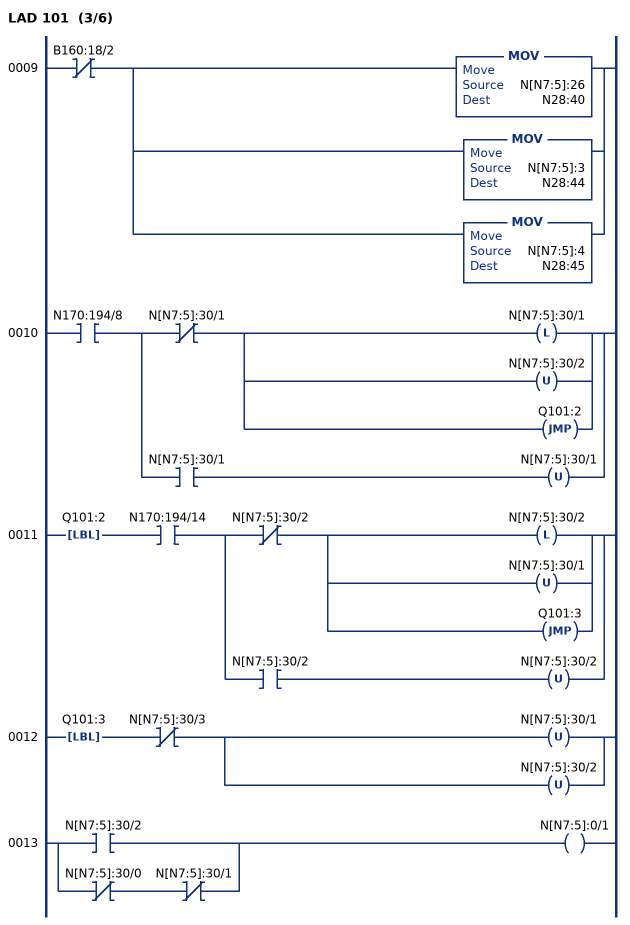
% Rung: 9 %
SOR XIO B160:18/2 BST MOV N[N7:5]:26 N28:40 NXB MOV N[N7:5]:3 N28:44 NXB MOV N[N7:5]:4 N28:45 BND EOR
% Rung: 10 %
SOR XIC N170:194/8 BST XIO N[N7:5]:30/1 BST OTL N[N7:5]:30/1 NXB OTU N[N7:5]:30/2 NXB JMP Q101:2 BND NXB XIC N[N7:5]:30/1 OTU N[N7:5]:30/1 BND EOR
% Rung: 11 %
SOR LBL Q101:2 XIC N170:194/14 BST XIO N[N7:5]:30/2 BST OTL N[N7:5]:30/2 NXB OTU N[N7:5]:30/1 NXB JMP Q101:3 BND NXB XIC N[N7:5]:30/2 OTU N[N7:5]:30/2 BND EOR
% Rung: 12 %
SOR LBL Q101:3 XIO N[N7:5]:30/3 BST OTU N[N7:5]:30/1 NXB OTU N[N7:5]:30/2 BND EOR
% Rung: 13 %
SOR BST XIC N[N7:5]:30/2 NXB XIO N[N7:5]:30/0 XIO N[N7:5]:30/1 BND OTE N[N7:5]:0/1 EOR

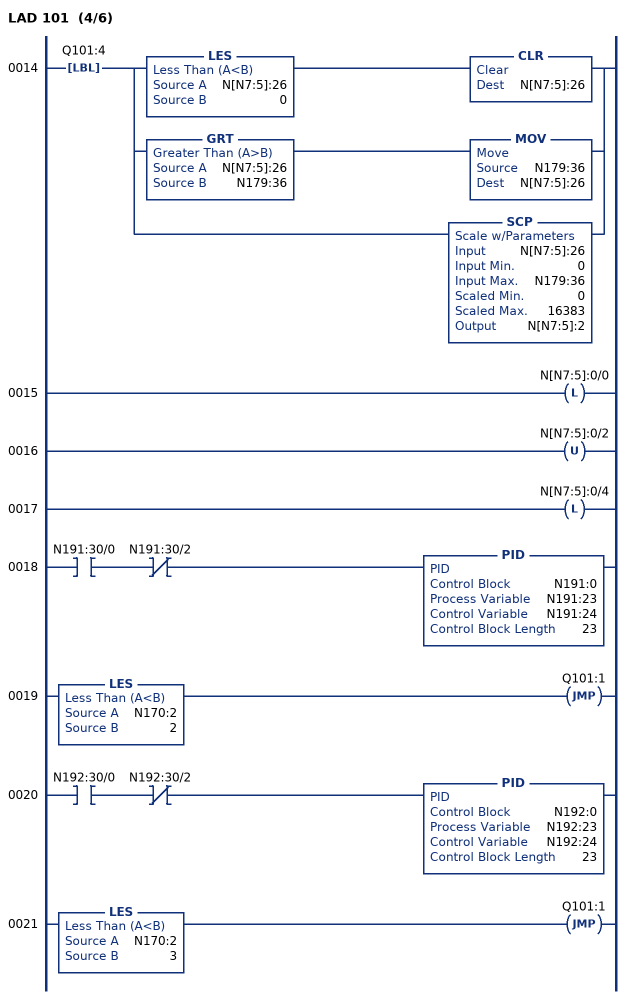
% Rung: 14 %
SOR LBL Q101:4 BST LES N[N7:5]:26 0 CLR N[N7:5]:26 NXB GRT N[N7:5]:26 N179:36 MOV N179:36 N[N7:5]:26 NXB SCP N[N7:5]:26 0 N179:36 0 16383 N[N7:5]:2 BND EOR
% Rung: 15 %
SOR OTL N[N7:5]:0/0 EOR
% Rung: 16 %
SOR OTU N[N7:5]:0/2 EOR
% Rung: 17 %
SOR OTL N[N7:5]:0/4 EOR
% Rung: 18 %
SOR XIC N191:30/0 XIO N191:30/2 PID N191:0 N191:23 N191:24 23 EOR
% Rung: 19 %
SOR LES N170:2 2 JMP Q101:1 EOR
% Rung: 20 %
SOR XIC N192:30/0 XIO N192:30/2 PID N192:0 N192:23 N192:24 23 EOR
% Rung: 21 %
SOR LES N170:2 3 JMP Q101:1 EOR

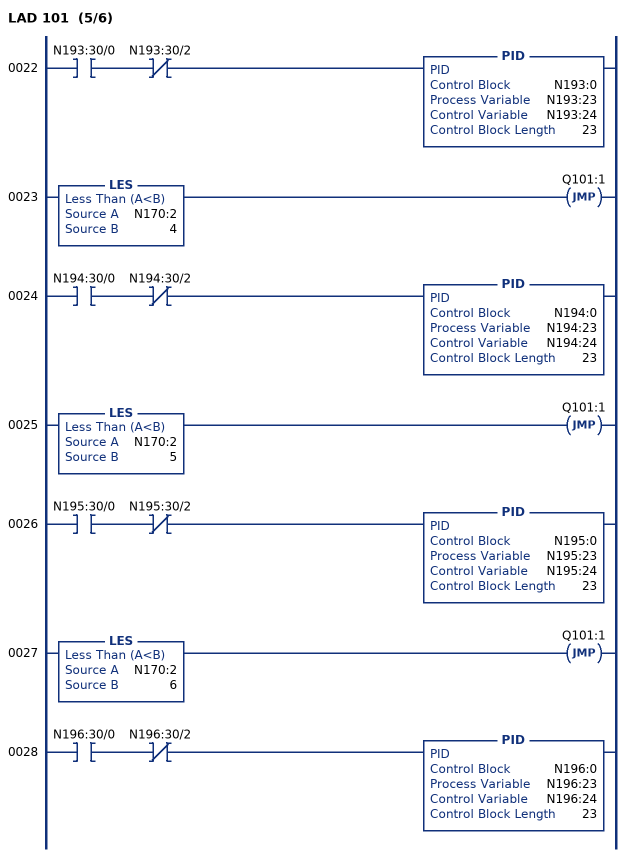
% Rung: 22 %
SOR XIC N193:30/0 XIO N193:30/2 PID N193:0 N193:23 N193:24 23 EOR
% Rung: 23 %
SOR LES N170:2 4 JMP Q101:1 EOR
% Rung: 24 %
SOR XIC N194:30/0 XIO N194:30/2 PID N194:0 N194:23 N194:24 23 EOR
% Rung: 25 %
SOR LES N170:2 5 JMP Q101:1 EOR
% Rung: 26 %
SOR XIC N195:30/0 XIO N195:30/2 PID N195:0 N195:23 N195:24 23 EOR
% Rung: 27 %
SOR LES N170:2 6 JMP Q101:1 EOR
% Rung: 28 %
SOR XIC N196:30/0 XIO N196:30/2 PID N196:0 N196:23 N196:24 23 EOR

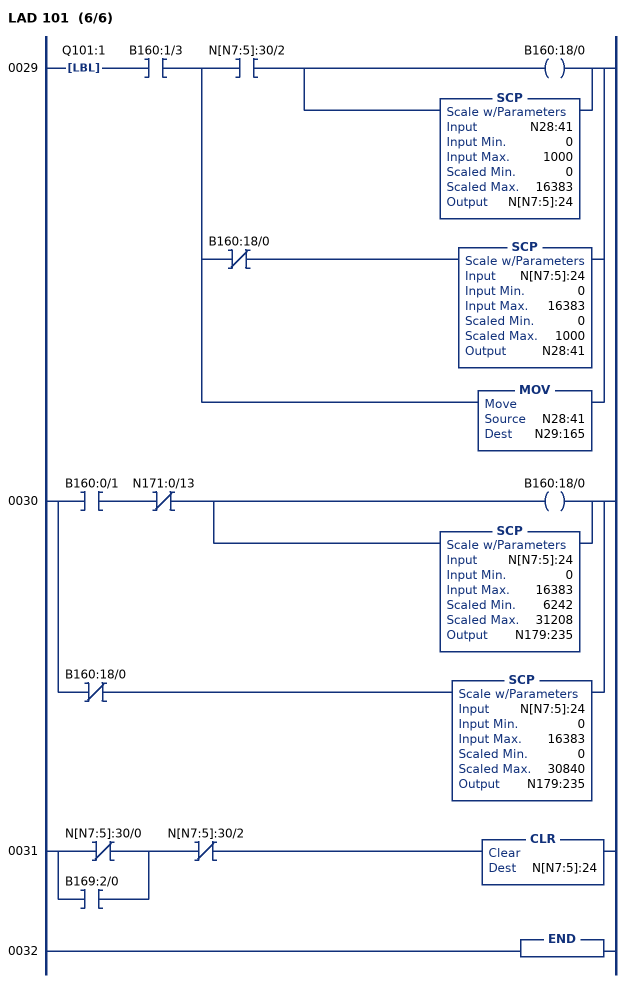
% Rung: 29 %
SOR LBL Q101:1 XIC B160:1/3 BST XIC N[N7:5]:30/2 BST OTE B160:18/0 NXB SCP N28:41 0 1000 0 16383 N[N7:5]:24 BND NXB XIO B160:18/0 SCP N[N7:5]:24 0 16383 0 1000 N28:41 NXB MOV N28:41 N29:165 BND EOR
% Rung: 30 %
SOR BST XIC B160:0/1 XIO N171:0/13 BST OTE B160:18/0 NXB SCP N[N7:5]:24 0 16383 6242 31208 N179:235 BND NXB XIO B160:18/0 SCP N[N7:5]:24 0 16383 0 30840 N179:235 BND EOR
% Rung: 31 %
SOR BST XIO N[N7:5]:30/0 NXB XIC B169:2/0 BND XIO N[N7:5]:30/2 CLR N[N7:5]:24 EOR
% Rung: 32 %
SOR END EOR

LADDER 102
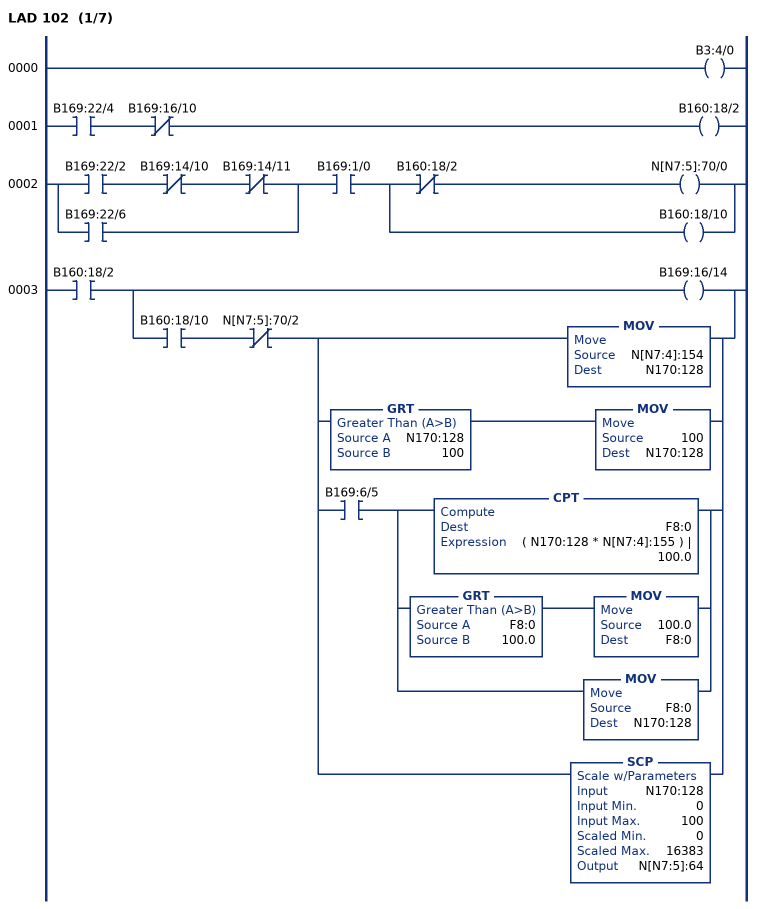
% Rung: 0 %
SOR OTE B3:4/0 EOR
% Rung: 1 %
SOR XIC B169:22/4 XIO B169:16/10 OTE B160:18/2 EOR
% Rung: 2 %
SOR BST XIC B169:22/2 XIO B169:14/10 XIO B169:14/11 NXB XIC B169:22/6 BND XIC B169:1/0 BST XIO B160:18/2 OTE N[N7:5]:70/0 NXB OTE B160:18/10 BND EOR
% Rung: 3 %
SOR XIC B160:18/2 BST OTE B169:16/14 NXB XIC B160:18/10 XIO N[N7:5]:70/2 BST BST MOV N[N7:4]:154 N170:128 NXB GRT N170:128 100 MOV 100 N170:128 BND NXB XIC B169:6/5 BST CPT F8:0 " ( N170:128 * N[N7:4]:155 ) | 100.0 " NXB GRT F8:0 100.0 MOV 100.0 F8:0 NXB MOV F8:0 N170:128 BND NXB SCP N170:128 0 100 0 16383 N[N7:5]:64 BND BND EOR

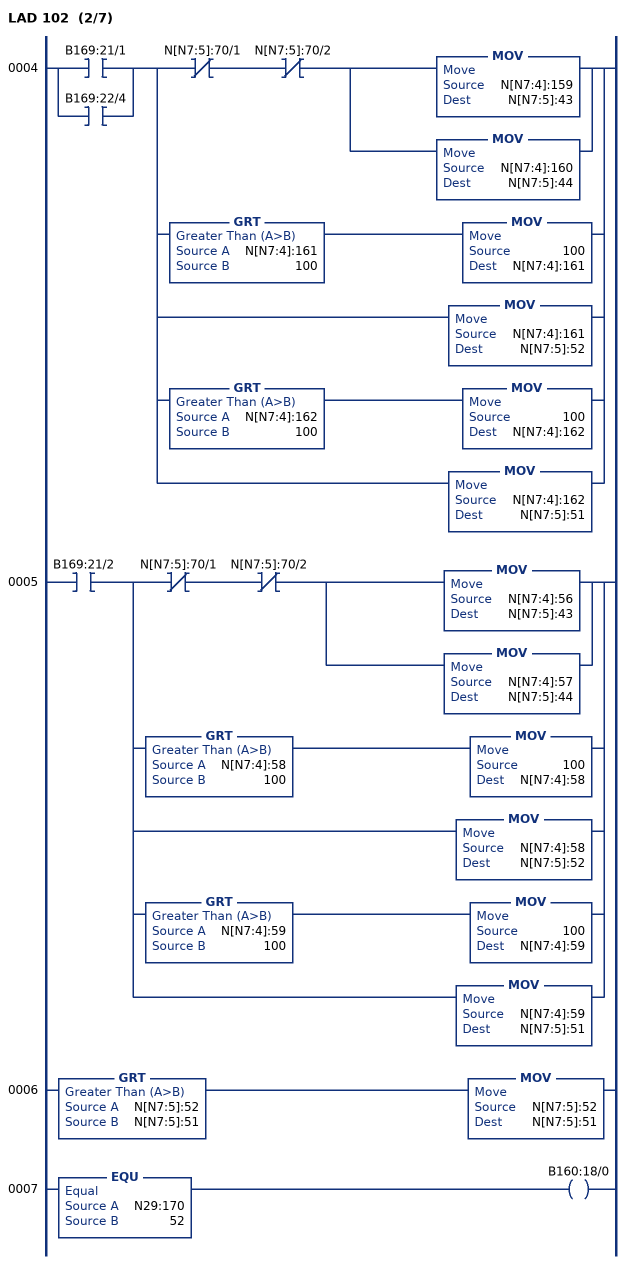
% Rung: 4 %
SOR BST XIC B169:21/1 NXB XIC B169:22/4 BND BST XIO N[N7:5]:70/1 XIO N[N7:5]:70/2 BST MOV N[N7:4]:159 N[N7:5]:43 NXB MOV N[N7:4]:160 N[N7:5]:44 BND NXB GRT N[N7:4]:161 100 MOV 100 N[N7:4]:161 NXB MOV N[N7:4]:161 N[N7:5]:52 NXB GRT N[N7:4]:162 100 MOV 100 N[N7:4]:162 NXB MOV N[N7:4]:162 N[N7:5]:51 BND EOR
% Rung: 5 %
SOR XIC B169:21/2 BST XIO N[N7:5]:70/1 XIO N[N7:5]:70/2 BST MOV N[N7:4]:56 N[N7:5]:43 NXB MOV N[N7:4]:57 N[N7:5]:44 BND NXB GRT N[N7:4]:58 100 MOV 100 N[N7:4]:58 NXB MOV N[N7:4]:58 N[N7:5]:52 NXB GRT N[N7:4]:59 100 MOV 100 N[N7:4]:59 NXB MOV N[N7:4]:59 N[N7:5]:51 BND EOR
% Rung: 6 %
SOR GRT N[N7:5]:52 N[N7:5]:51 MOV N[N7:5]:52 N[N7:5]:51 EOR
% Rung: 7 %
SOR EQU N29:170 52 OTE B160:18/0 EOR

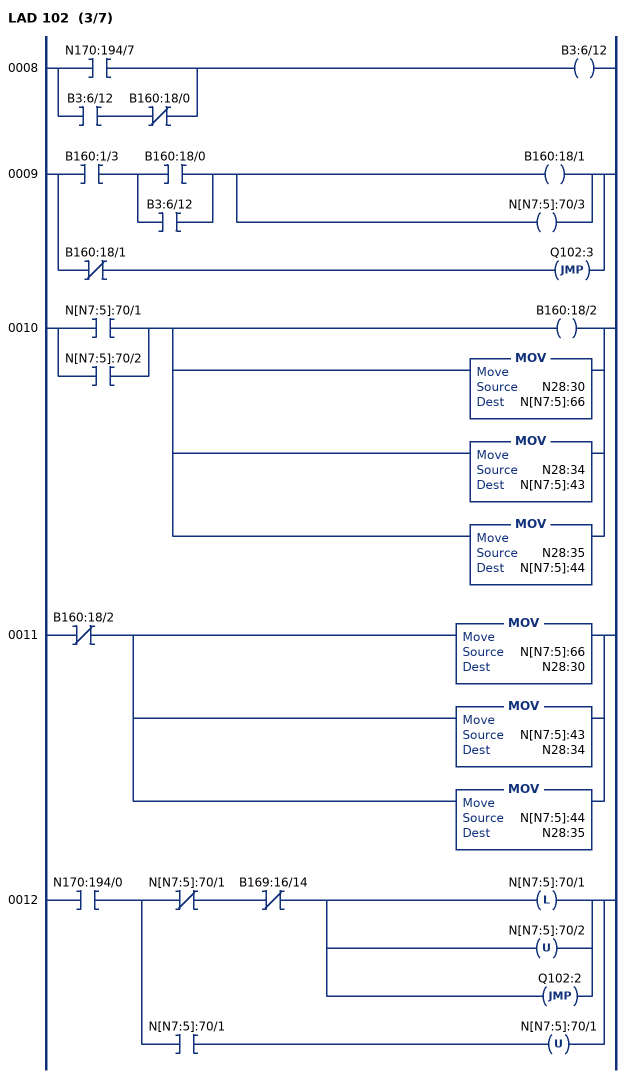
% Rung: 8 %
SOR BST XIC N170:194/7 NXB XIC B3:6/12 XIO B160:18/0 BND OTE B3:6/12 EOR
% Rung: 9 %
SOR BST XIC B160:1/3 BST XIC B160:18/0 NXB XIC B3:6/12 BND BST OTE B160:18/1 NXB OTE N[N7:5]:70/3 BND NXB XIO B160:18/1 JMP Q102:3 BND EOR
% Rung: 10 %
SOR BST XIC N[N7:5]:70/1 NXB XIC N[N7:5]:70/2 BND BST OTE B160:18/2 NXB MOV N28:30 N[N7:5]:66 NXB MOV N28:34 N[N7:5]:43 NXB MOV N28:35 N[N7:5]:44 BND EOR
% Rung: 11 %
SOR XIO B160:18/2 BST MOV N[N7:5]:66 N28:30 NXB MOV N[N7:5]:43 N28:34 NXB MOV N[N7:5]:44 N28:35 BND EOR
% Rung: 12 %
SOR XIC N170:194/0 BST XIO N[N7:5]:70/1 XIO B169:16/14 BST OTL N[N7:5]:70/1 NXB OTU N[N7:5]:70/2 NXB JMP Q102:2 BND NXB XIC N[N7:5]:70/1 OTU N[N7:5]:70/1 BND EOR

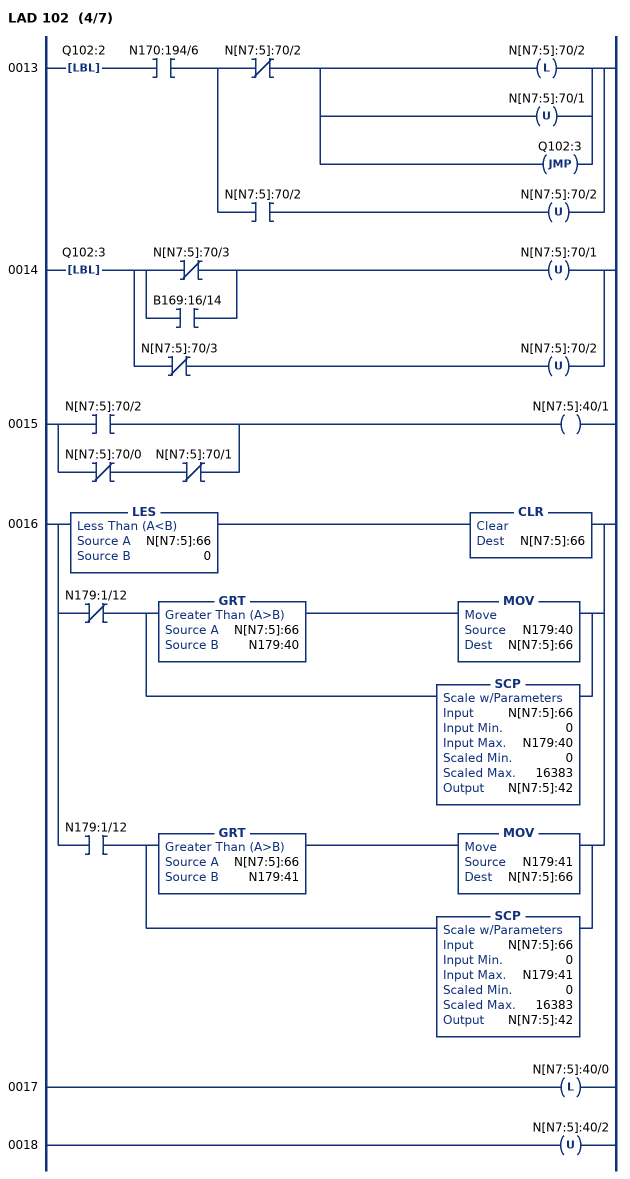
% Rung: 13 %
SOR LBL Q102:2 XIC N170:194/6 BST XIO N[N7:5]:70/2 BST OTL N[N7:5]:70/2 NXB OTU N[N7:5]:70/1 NXB JMP Q102:3 BND NXB XIC N[N7:5]:70/2 OTU N[N7:5]:70/2 BND EOR
% Rung: 14 %
SOR LBL Q102:3 BST BST XIO N[N7:5]:70/3 NXB XIC B169:16/14 BND OTU N[N7:5]:70/1 NXB XIO N[N7:5]:70/3 OTU N[N7:5]:70/2 BND EOR
% Rung: 15 %
SOR BST XIC N[N7:5]:70/2 NXB XIO N[N7:5]:70/0 XIO N[N7:5]:70/1 BND OTE N[N7:5]:40/1 EOR
% Rung: 16 %
SOR BST LES N[N7:5]:66 0 CLR N[N7:5]:66 NXB XIO N179:1/12 BST GRT N[N7:5]:66 N179:40 MOV N179:40 N[N7:5]:66 NXB SCP N[N7:5]:66 0 N179:40 0 16383 N[N7:5]:42 BND NXB XIC N179:1/12 BST GRT N[N7:5]:66 N179:41 MOV N179:41 N[N7:5]:66 NXB SCP N[N7:5]:66 0 N179:41 0 16383 N[N7:5]:42 BND BND EOR
% Rung: 17 %
SOR OTL N[N7:5]:40/0 EOR
% Rung: 18 %
SOR OTU N[N7:5]:40/2 EOR

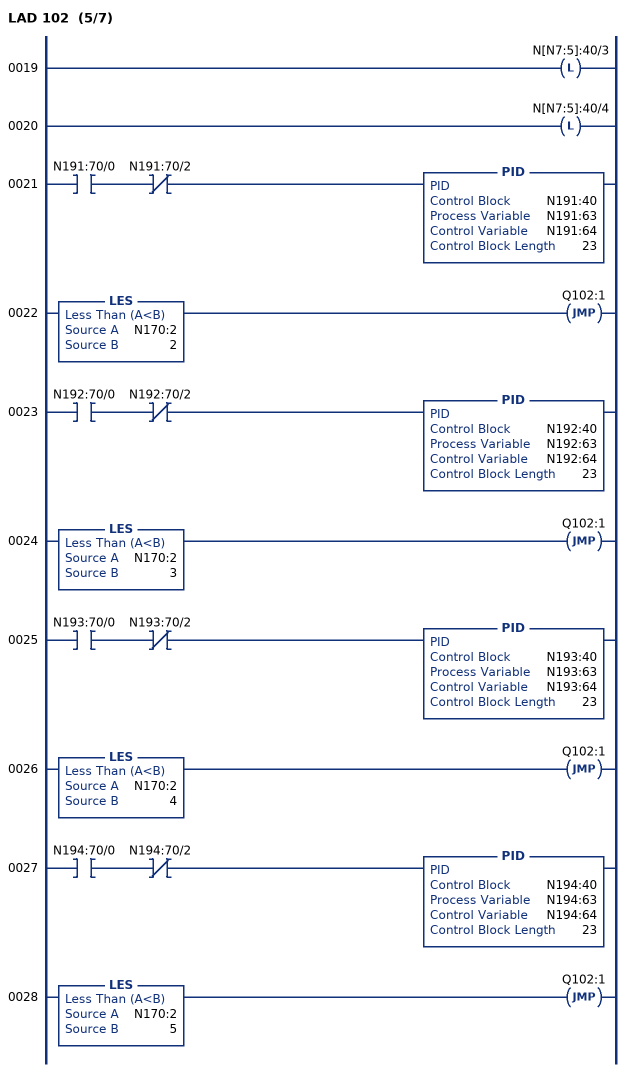
% Rung: 19 %
SOR OTL N[N7:5]:40/3 EOR
% Rung: 20 %
SOR OTL N[N7:5]:40/4 EOR
% Rung: 21 %
SOR XIC N191:70/0 XIO N191:70/2 PID N191:40 N191:63 N191:64 23 EOR
% Rung: 22 %
SOR LES N170:2 2 JMP Q102:1 EOR
% Rung: 23 %
SOR XIC N192:70/0 XIO N192:70/2 PID N192:40 N192:63 N192:64 23 EOR
% Rung: 24 %
SOR LES N170:2 3 JMP Q102:1 EOR
% Rung: 25 %
SOR XIC N193:70/0 XIO N193:70/2 PID N193:40 N193:63 N193:64 23 EOR
% Rung: 26 %
SOR LES N170:2 4 JMP Q102:1 EOR
% Rung: 27 %
SOR XIC N194:70/0 XIO N194:70/2 PID N194:40 N194:63 N194:64 23 EOR
% Rung: 28 %
SOR LES N170:2 5 JMP Q102:1 EOR

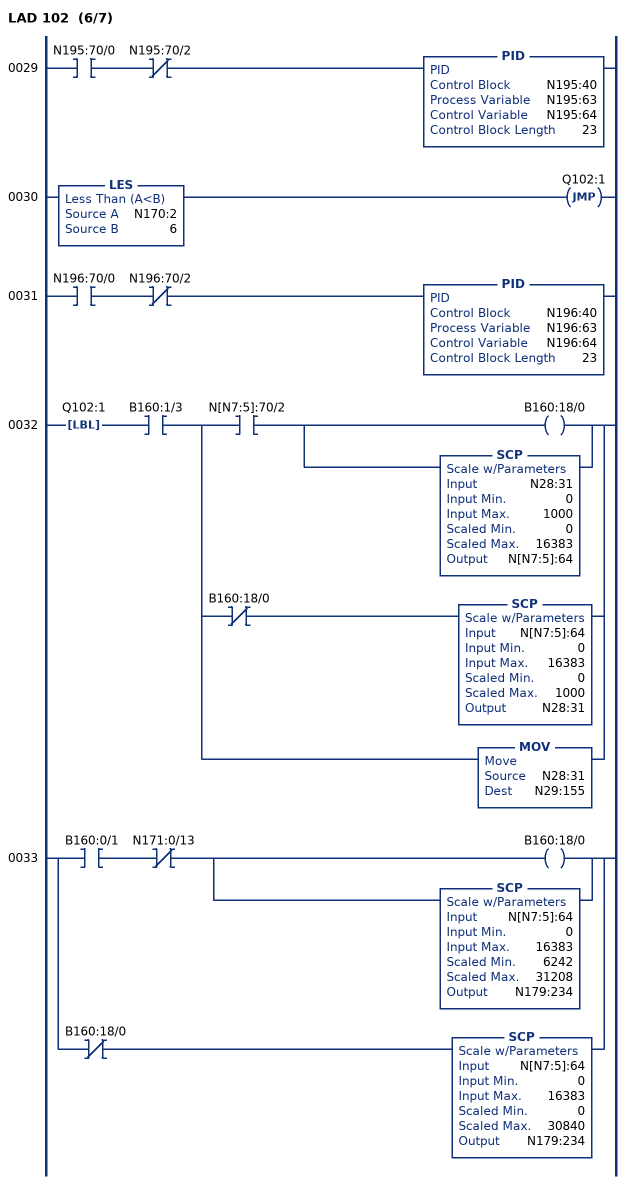
% Rung: 29 %
SOR XIC N195:70/0 XIO N195:70/2 PID N195:40 N195:63 N195:64 23 EOR
% Rung: 30 %
SOR LES N170:2 6 JMP Q102:1 EOR
% Rung: 31 %
SOR XIC N196:70/0 XIO N196:70/2 PID N196:40 N196:63 N196:64 23 EOR
% Rung: 32 %
SOR LBL Q102:1 XIC B160:1/3 BST XIC N[N7:5]:70/2 BST OTE B160:18/0 NXB SCP N28:31 0 1000 0 16383 N[N7:5]:64 BND NXB XIO B160:18/0 SCP N[N7:5]:64 0 16383 0 1000 N28:31 NXB MOV N28:31 N29:155 BND EOR
% Rung: 33 %
SOR BST XIC B160:0/1 XIO N171:0/13 BST OTE B160:18/0 NXB SCP N[N7:5]:64 0 16383 6242 31208 N179:234 BND NXB XIO B160:18/0 SCP N[N7:5]:64 0 16383 0 30840 N179:234 BND EOR

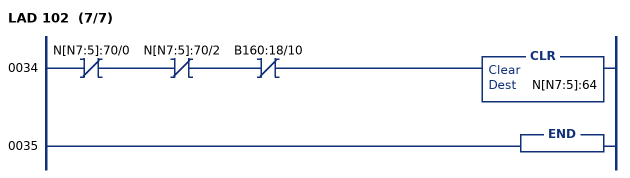
% Rung: 34 %
SOR XIO N[N7:5]:70/0 XIO N[N7:5]:70/2 XIO B160:18/10 CLR N[N7:5]:64 EOR
% Rung: 35 %
SOR END EOR

DATA TABLE (non-zero values as saved)
DATA B3
% B3:0 % 0X0802 0X0000 0X0200 0X0000 0X0009 0X0084 0X8000 0X0000 0X0040 0X0000
% B3:10 % 0X0000 0X0000 0X0000 0X0000 0X0000 0X0000 0X0000 0X0001
DATA T4
% .PRE .ACC %
% T4:2 % 5 5
% T4:3 % 5 0
% T4:9 % 60 0
% T4:10 % 2 0
% T4:11 % 3 0
% T4:15 % 5 0
% T4:19 % 1 0
% T4:20 % 1200 0
% T4:21 % 15 0
% T4:22 % 15 0
% T4:23 % 15 0
% T4:24 % 3 0
% T4:25 % 3 0
% T4:26 % 3 0
% T4:27 % 2 0
% T4:28 % 2 0
% T4:30 % 50 50
% T4:31 % 50 50
% T4:32 % 50 50
% T4:33 % 15 0
% T4:34 % 15 0
% T4:35 % 110 0
% T4:36 % 20 0
DATA C5
% .PRE .ACC %
% C5:5 % 3 0
DATA R6
% .LEN .POS %
% R6:0 % 16 0
% R6:1 % 10 0
% R6:2 % 10 0
% R6:3 % 10 0
% R6:4 % 10 0
% R6:5 % 10 0
% R6:6 % 10 0
% R6:7 % 11 0
% R6:8 % 8 0
% R6:9 % 16 0
% R6:11 % 10 10
% R6:12 % 10 10
% R6:13 % 10 0
% R6:14 % 10 0
% R6:15 % 10 0
% R6:16 % 10 0
% R6:17 % 32 0
% R6:18 % 6 0
% R6:19 % 6 0
% R6:20 % 32 0
DATA N7
% N7:0 % 2 162 172 182 60 192 202 212 232 0
% N7:10 % 41 1 166 0 0 0 0 0 0 0
% N7:20 % 3 5 1 0 0 0 0 0 0 0
% N7:30 % 0 8 0 2 0 -32768 0 0 0 0
% N7:40 % -32768 0 0 0 0 0 0 0 0 0
% N7:60 % 0 2 0 0 0 0 0 0 0 0
% N7:100 % 150 41 40 63 100 0 41 10 0 0
% N7:110 % 44 0 63 0 0 0 38 1 38 1
% N7:120 % 0 38 1 0 3 15 3 40 70 100
% N7:130 % 0 0 0 -1 0
DATA T10
% .PRE .ACC %
% T10:0 % 12 0
% T10:1 % 12 0
% T10:2 % 12 0
% T10:3 % 3 0
DATA N11
% N11:0 % 0 1 4 21 31 0 0 0 0 0
% N11:10 % 0 81 91 0 0 0 1 4 0 0
% N11:20 % 41 51 0 0 0 0 81 91 0 0
% N11:30 % 0 1 4 21 31 41 51 0 0 0
% N11:40 % 0 81 91 0 0 0 1 4 0 0
% N11:50 % 41 51 21 31 0 0 81 91 0 0
% N11:60 % 0 1 4 21 31 41 51 21 31 0
% N11:70 % 0 81 91 0 0 0 1 4 21 31
% N11:80 % 0 0 0 0 61 0 81 91 0 0
% N11:90 % 0 1 4 21 31 41 51 0 0 61
% N11:100 % 0 81 91 0 0 0 1 4 0 0
% N11:110 % 41 51 21 31 61 0 81 91 0 0
% N11:120 % 0 1 4 21 31 0 0 0 0 0
% N11:130 % 71 153 91 0 0 0 1 4 21 31
% N11:140 % 41 51 0 0 0 71 153 91 0 0
% N11:160 % 71 91 0 0 0 0 1 4 0 0
% N11:170 % 0 0 0 0 0 0 81 91 0 0
% N11:190 % 71 153 91 0 0 0 0 0 0 0
% N11:200 % 0 0 0 0 61 0 81 91 0 0
DATA N12
% N12:0 % 0 101 105 135 0 0 101 125 135 0
% N12:10 % 0 101 141 135 0 0 101 115 135 0
% N12:20 % 0 101 127 135 0 0 101 161 135 0
% N12:30 % 0 101 129 135 0 0 101 181 135 0
% N12:40 % 0 101 201 135 0 0 101 131 135 0
% N12:50 % 0 101 195 135 0
DATA N14
% N14:0 % 0 8193 0 0 8192 8240 8192 8240 48 0
% N14:10 % 528 562 34 1 48 34 0 0 0 0
% N14:20 % 0 1 40 0 40 2088 2600 -30174 2602 2082
% N14:30 % 0 2049 0 -30688 2048 -30688 -30688 -28640 -32222 4130
% N14:40 % 0 1 36 0 36 1060 1572 -31198 1574 1058
% N14:50 % 0 1025 0 -31712 1024 -31712 -31712 -28640 -32222 4130
% N14:60 % 0 1 -32736 0 -32736 -32224 -32222 2 0 0
% N14:70 % 0 2 32 0 32 544 0 546 34 0
% N14:80 % 0 1 0 -28640 4096 -28640 -28640 -28640 0 0
% N14:90 % 0 4096 0 0 0 0 0 0 0 0
% N14:100 % 0 193 0 0 0 -30496 2281 2280 2280 2280
% N14:110 % 2280 -30528 0 0 0 -31520 1253 1252 1252 1252
% N14:120 % 1252 -31552 0 0 0 200 0 196 0 208
% N14:130 % 0 192 0 0 0 -32640 -32576 0 0 0
% N14:140 % 0 2256 456 200 132 2276 488 201 -32640 -30528
% N14:150 % 456 201 0 1 -32768 0 -32768 -32768 -32254 2
% N14:160 % 0 1232 452 196 136 1256 484 197 -32640 -31552
% N14:170 % 452 197 0 0 0 0 0 0 0 0
% N14:180 % 0 -28480 464 208 136 4328 496 209 -32640 -28480
% N14:190 % 464 209 0 0 0 -32576 0 0 0 0
% N14:200 % 0 -28480 464 208 132 4324 496 209 -32640 -28480
% N14:210 % 464 209
DATA N15
% N15:0 % 0 0 0 0 0 1 0 1 1 0
% N15:10 % 1 1 1 0 1 1 0 0 0 0
% N15:20 % 0 0 1 0 1 1 1 1 1 1
% N15:30 % 0 0 0 1 0 1 1 1 1 1
% N15:40 % 0 0 1 0 1 1 1 1 1 1
% N15:50 % 0 0 0 1 0 1 1 1 1 1
% N15:60 % 0 0 1 0 1 1 1 1 0 0
% N15:70 % 0 1 17 0 17 49 0 49 33 0
% N15:80 % 0 0 0 1 0 1 1 1 0 0
% N15:100 % 0 0 0 0 0 5 1 1 1 5
% N15:110 % 1 1 0 0 0 3 1 1 1 3
% N15:120 % 1 1 0 0 0 385 0 385 0 1
% N15:130 % 0 17 0 0 0 384 385 0 0 0
% N15:140 % 0 1 1 1 0 1 1 1 0 1
% N15:150 % 1 1 0 32 33 32 33 1 1 1
% N15:160 % 0 1 1 1 0 1 1 1 0 1
% N15:170 % 1 1 0 0 0 0 0 0 0 0
% N15:180 % 0 1 1 1 0 1 1 1 0 1
% N15:190 % 1 1 0 0 0 33 0 0 0 0
% N15:200 % 0 1 1 1 0 1 1 1 0 1
% N15:210 % 1 1
DATA N16
% N16:0 % 1 0 0 0 0 2048 2048 2048 2048 2048
% N16:10 % 8 8 8 8 8 8 1 1 1 1
% N16:20 % 1 128 2 2 2 2 2 2 2 2
% N16:30 % 1 16 0 16 16 16 16 16 16 16
% N16:40 % 1 128 4 4 4 4 4 4 4 4
% N16:50 % 1 32 0 32 32 32 32 32 32 32
% N16:60 % 1 128 128 128 128 128 128 128 1 1
% N16:70 % 1 256 256 256 256 256 1 256 256 1
% N16:80 % 1 64 0 64 64 64 64 64 1 1
% N16:90 % 1 1 1 1 1 1 1 1 1 1
% N16:100 % 1 1 1 1 1 512 512 512 512 512
% N16:110 % 512 1 1 1 1 1024 1024 1024 1024 1024
% N16:120 % 1024 1 1 1 1 1 1 1 1 1
% N16:130 % 1 1 1 1 1 1 1 1 1 1
% N16:140 % 1 1 1 1 1 16384 16384 1 1 1
% N16:150 % 1 1 1 1 1 1 1 1 1 1
% N16:160 % 1 1 1 1 1 8192 8192 1 1 1
% N16:170 % 1 1 1 1 1 1 1 1 1 1
% N16:180 % 1 1 1 1 1 8192 8192 1 1 1
% N16:190 % 1 1 1 1 1 1 1 1 1 1
% N16:200 % 1 1 1 1 1 16384 16384 1 1 1
% N16:210 % 1 1
DATA N17
% N17:0 % 0 0 0 0 211 -8 195 104 165 195
% N17:10 % 0 182 60 0 168 60 0 0 0 0
% N17:20 % 0 0 103 195 104 203 61 -3 -2 60
% N17:30 % 0 0 0 103 195 104 204 169 193 60
% N17:40 % 0 0 103 195 104 203 62 -3 -1 60
% N17:50 % 0 0 0 103 195 104 204 169 193 60
% N17:60 % 0 0 103 195 104 0 183 60 0 0
% N17:70 % 0 60 103 195 104 61 0 194 60 0
% N17:80 % 0 0 0 103 195 104 167 208 0 0
% N17:90 % 0 195 0 0 0 0 0 0 0 0
% N17:100 % 0 0 0 0 0 10082 10 11 11082 11083
% N17:110 % 10087 -4 0 0 0 10083 20 21 11082 11083
% N17:120 % 10087 -4 0 0 0 10093 0 10093 0 10093
% N17:130 % 0 10093 0 0 0 10095 53 0 0 0
% N17:140 % 0 28 33 10093 10095 28 34 10093 10095 28
% N17:150 % 35 10093 0 0 103 195 104 169 193 60
% N17:160 % 0 28 33 10093 10095 28 34 10093 10095 28
% N17:170 % 35 10093 0 0 0 0 0 0 0 0
% N17:180 % 0 28 33 10093 10095 28 34 10093 10095 28
% N17:190 % 35 10093 0 0 0 0 0 0 0 0
% N17:200 % 0 28 33 10093 10095 28 34 10093 10095 28
% N17:210 % 35 10093
DATA N18
% N18:0 % 0 10081 0 0 0 0 10097 0 0 10097
% N18:10 % 10081 -5 0 10081 0 0 0 0 0 0
% N18:20 % 0 10081 0 10097 0 105 10081 0 -5 0
% N18:30 % 0 10081 0 0 10097 0 105 0 0 0
% N18:40 % 0 10081 0 10097 0 105 10081 0 -5 0
% N18:50 % 0 10081 0 0 10097 0 105 0 0 0
% N18:60 % 0 10081 0 10097 0 10081 -5 0 0 0
% N18:70 % 0 0 0 10097 0 10081 0 0 0 0
% N18:80 % 0 10081 0 0 10097 0 0 170 0 0
% N18:90 % 0 10097 0 0 0 0 0 0 0 0
% N18:100 % 0 10081 0 0 0 -6 0 0 0 11084
% N18:110 % 10088 0 0 0 0 -6 0 0 0 11084
% N18:120 % 10088 0 0 0 0 10094 0 10094 0 10094
% N18:130 % 0 10094 0 0 0 0 0 0 0 0
% N18:140 % 0 0 0 10104 0 0 -7 10104 0 0
% N18:150 % 0 10104 0 10081 0 10097 0 0 0 0
% N18:160 % 0 0 0 10104 0 0 -7 10104 0 0
% N18:170 % 0 10104 0 0 0 0 0 0 0 0
% N18:180 % 0 0 0 10104 0 0 -7 10104 0 0
% N18:190 % 0 10104 0 0 0 0 0 0 0 0
% N18:200 % 0 0 0 10104 0 0 -7 10104 0 0
% N18:210 % 0 10104
DATA N19
% N19:0 % 0 128 0 0 1 2 256 2 2 256
% N19:10 % 128 512 32 128 2 32 0 0 0 0
% N19:20 % 0 128 2 256 2 2048 64 2 8192 32
% N19:30 % 0 128 0 2 256 2 1024 2 1 32
% N19:40 % 0 128 2 256 2 2048 64 2 8192 32
% N19:50 % 0 128 0 2 256 2 1024 2 1 32
% N19:60 % 0 128 2 256 2 128 512 32 0 0
% N19:70 % 0 32 2 256 2 64 0 512 32 0
% N19:80 % 0 128 0 2 256 2 2 1024 0 0
% N19:90 % 0 256 0 0 0 0 0 0 0 0
% N19:100 % 0 128 0 0 0 4 1 1 1 1
% N19:110 % 512 2 0 0 0 8 1 1 1 1
% N19:120 % 512 2 0 0 0 256 0 256 0 256
% N19:130 % 0 256 0 0 0 1 2 0 0 0
% N19:140 % 0 2 1 256 1 2 512 256 1 2
% N19:150 % 1 256 0 128 2 256 2 2 1 32
% N19:160 % 0 2 1 256 1 2 512 256 1 2
% N19:170 % 1 256 0 0 0 0 0 0 0 0
% N19:180 % 0 2 1 256 1 2 512 256 1 2
% N19:190 % 1 256 0 0 0 16384 0 0 0 0
% N19:200 % 0 2 1 256 1 2 512 256 1 2
% N19:210 % 1 256
DATA N20
% N20:0 % 0 1 0 0 2 2 2 2 2 2
% N20:10 % 2 2 2 2 2 2 1 1 1 1
% N20:20 % 1 1 4 4 4 4 4 4 4 4
% N20:30 % 1 4 0 4 4 4 4 1 1 1
% N20:40 % 1 1 8 8 8 8 8 8 8 8
% N20:50 % 1 8 0 8 8 8 8 1 1 1
% N20:60 % 1 32 32 32 32 32 32 32 1 1
% N20:70 % 1 16 16 16 16 16 1 16 16 1
% N20:80 % 1 64 0 64 64 64 64 64 1 1
% N20:90 % 1 1 1 1 1 1 1 1 1 1
% N20:100 % 1 1 1 1 1 4 4 4 4 4
% N20:110 % 4 4 1 1 1 8 8 8 8 8
% N20:120 % 8 8 1 1 1 4 4 8 8 1
% N20:130 % 1 1 1 1 1 1 1 1 1 1
% N20:140 % 1 1 1 1 1 1 1 1 1 1
% N20:150 % 1 1 1 16 16 16 16 1 1 1
% N20:160 % 1 1 1 1 1 1 1 1 1 1
% N20:170 % 1 1 1 1 1 1 1 1 1 1
% N20:180 % 1 1 1 1 1 1 1 1 1 1
% N20:190 % 1 1 1 1 1 1 1 1 1 1
% N20:200 % 1 1 1 1 1 1 1 1 1 1
% N20:210 % 1 1
DATA N21
% N21:0 % 0 1 0 0 4 4 4 4 1 1
% N21:10 % 1 32 1 1 1 1 1 1 1 1
% N21:20 % 1 1 1 1 1 4 1 2 32 8
% N21:30 % 1 8 0 8 8 8 16 1 32 1
% N21:40 % 1 1 1 1 1 4 1 2 32 8
% N21:50 % 1 8 0 8 8 8 16 1 32 1
% N21:60 % 1 1 1 1 1 1 32 1 1 1
% N21:70 % 1 1 1 1 1 1 1 32 1 1
% N21:80 % 1 1 0 1 1 1 32 16 1 1
% N21:90 % 1 1 1 1 1 1 1 1 1 1
% N21:100 % 1 1 1 1 1 256 1 1 512 1024
% N21:110 % 1 2048 1 1 1 256 1 1 512 1024
% N21:120 % 1 2048 1 1 1 4096 1 4096 1 4096
% N21:130 % 1 4096 1 1 1 1 1 1 1 1
% N21:140 % 1 1 1 1 1 1 1 1 1 1
% N21:150 % 1 1 1 1 1 1 1 1 32 1
% N21:160 % 1 1 1 1 1 1 1 1 1 1
% N21:170 % 1 1 1 1 1 1 1 1 1 1
% N21:180 % 1 1 1 1 1 1 1 1 1 1
% N21:190 % 1 1 1 1 1 4 1 1 1 1
% N21:200 % 1 1 1 1 1 1 1 1 1 1
% N21:210 % 1 1
DATA N22
% N22:0 % 0 529 0 0 144 16 144 16 -32768 128
% N22:10 % 256 -32512 258 2 -32766 1 0 0 0 0
% N22:20 % 0 1040 0 128 0 2048 256 1024 -32736 257
% N22:30 % 0 0 0 8192 8320 8192 8192 -8192 -32768 1
% N22:40 % 0 1040 0 128 0 2048 256 1024 -32736 257
% N22:50 % 0 0 0 8192 8320 8192 8192 -8192 -32768 1
% N22:60 % 0 532 20 148 20 0 -32768 1 0 0
% N22:70 % 0 0 0 128 0 256 0 -32768 257 0
% N22:80 % 0 16 16 8208 8336 8208 -8192 -32767 0 0
% N22:90 % 0 193 0 0 0 0 0 0 0 0
% N22:100 % 0 513 0 0 0 0 0 4096 4096 4096
% N22:110 % 0 1 0 0 0 0 0 4096 4096 4096
% N22:120 % 0 1 0 0 0 9 0 9 0 9
% N22:130 % 0 9 0 0 0 0 1 0 0 0
% N22:140 % 0 0 0 8 0 0 0 8 0 0
% N22:150 % 0 9 0 0 0 128 0 -32768 -32768 1
% N22:160 % 0 0 0 8 0 0 0 8 0 0
% N22:170 % 0 9 0 0 0 0 0 0 0 0
% N22:180 % 0 0 0 8 0 0 0 8 0 0
% N22:190 % 0 9 0 0 0 1 0 0 0 0
% N22:200 % 0 0 0 8 0 0 0 8 0 0
% N22:210 % 0 9
DATA N23
% N23:0 % 0 146 0 0 6 10 0 0 66 0
% N23:10 % 1 1 1 0 0 0 0 0 0 0
% N23:20 % 0 0 2 10 2 2 0 0 2 0
% N23:30 % 0 0 0 2 10 2 2 0 0 0
% N23:40 % 0 0 2 10 2 2 0 0 2 0
% N23:50 % 0 0 0 2 10 2 2 0 0 0
% N23:80 % 0 0 0 0 0 0 2 2 0 0
DATA N24
% N24:0 % 0 8 0 0 8 8 8 8 8 8
% N24:10 % 8 2 32 8 8 32 1 1 1 1
% N24:20 % 1 8 8 8 8 8 16 2 2 32
% N24:30 % 1 8 0 8 8 8 8 8 2 32
% N24:40 % 1 8 8 8 8 8 16 2 2 32
% N24:50 % 1 8 0 8 8 8 8 8 2 32
% N24:60 % 1 8 8 8 8 8 8 32 1 1
% N24:70 % 1 32 8 8 8 16 1 2 32 1
% N24:80 % 1 8 0 8 8 8 8 8 1 1
% N24:90 % 1 1 1 1 1 1 1 1 1 1
% N24:100 % 1 8 1 1 1 8 8 8 8 8
% N24:110 % 8 8 1 1 1 8 8 8 8 8
% N24:120 % 8 8 1 1 1 1 1 1 1 1
% N24:130 % 1 1 1 1 1 8 8 1 1 1
% N24:140 % 1 8 1 1 1 1 1 8 8 8
% N24:150 % 1 8 0 8 8 8 8 8 2 32
% N24:160 % 0 8 1 1 1 1 1 8 8 8
% N24:170 % 1 8 0 0 0 0 0 0 0 0
% N24:180 % 0 8 1 1 1 1 1 8 8 8
% N24:190 % 1 8 0 0 0 8 0 0 0 0
% N24:200 % 0 8 1 1 1 1 1 8 8 8
% N24:210 % 1 8
DATA B25
% B25:0 % 0X0000 0X0020 0X0000 0X0000 0X0000 0X0000 0X0000 0X0000 0X0000 0X0001
DATA N28
% N28:10 % 0 1 1 1 1 141 1 1 141 2
% N28:20 % 0 141 1923 7 12 17 0 50 1 0
% N28:30 % 2000 0 0 0 160 20 0 0 0 0
% N28:40 % 500 0 0 0 100 5 0 0 0 0
% N28:100 % 0 0 60 140 200 150 5 242 80 16
% N28:110 % 100 27 20 20 350 330 2 3 5 5
% N28:120 % 5 5 5 5 0 0 0 0 0 0
DATA N29
% N29:0 % 0 0 512 0 0 0 -242 -1 512 6144
% N29:60 % 16 0 0 0 0 0 16 0 0 0
% N29:70 % 0 0 1 0 0 0 0 0 16 0
% N29:80 % 0 0 0 0 16 0 0 0 0 0
% N29:90 % 32 0 0 0 0 0 0 0 0 0
% N29:100 % 0 0 0 16 4 5 0 0 0 0
% N29:110 % 142 0 0 0 0 0 1 0 0 0
% N29:120 % 1 0 0 0 0 0 0 0 1 1923
% N29:130 % 7 12 17 0 50 0 0 0 0 0
% N29:140 % 303 0 303 0 0 6 0 6 0 0
% N29:150 % 3 3 0 0 0 0 70 15 0 0
% N29:160 % 372 372 0 0 0 0 250 50 0 0
% N29:170 % 2 0 0 0 0 0 0 0 0 0
% N29:180 % 222 10601 0 0 0 0 0 0 0 0
% N29:190 % 291 2 23 303 3 6 132 0 1 113
% N29:200 % 0 0 111 3 0 109 3 0 1 0
DATA N38
% N38:0 % 0 2000 800 10 5 5 0 0 480 60
% N38:10 % 480 180 270 135 20 953 0 0 3610 50
% N38:20 % 480 180 500 133 14 858 60 3 0 0
% N38:30 % 1 0 0 0 0 0 0 0 0 0
DATA N39
% N39:0 % 0 80 120 200 100 5 160 20 1 100
% N39:10 % 27 20 20 350 330 2 3 5 5 5
% N39:20 % 5 5 5 3 1 0 0 0 0 0
% N39:40 % 0 60 140 200 150 5 242 80 16 100
% N39:50 % 27 20 20 350 330 2 3 5 5 5
% N39:60 % 5 5 5 0 0 0 0 0 0 0
DATA N40
% N40:0 % 0 2000 800 10 5 5 0 0 480 60
% N40:10 % 480 180 270 135 20 953 0 0 3610 50
% N40:20 % 480 180 500 133 14 858 60 3 0 0
% N40:30 % 1 0 0 0 0 0 0 0 0 0
% N40:50 % 0 80 120 200 100 5 160 20 1 100
% N40:60 % 27 20 20 350 330 2 3 5 5 5
% N40:70 % 5 5 5 3 1 0 0 0 0 0
% N40:100 % 0 3 20003 460 0 162 0 0 0 0
% N40:150 % 0 0 0 0 1500 100 750 300 15 90
% N40:160 % 15 0 100 0 0 800 0 600 800 900
% N40:170 % 60 30 55 60 30 60 30 95 0 0
% N40:180 % 10 600 0 600 600 600 600 600 300 300
% N40:190 % 300 300 300 0 600 30 30 300 50 60
% N40:200 % 40 60 40 5 5 70 30 20 5 50
% N40:210 % 50 0 0 0 0 0 0 0 0 0
DATA N41
% N41:0 % 1 0 20201 0 0 0 0 0 0 0
% N41:10 % 0 1 20201 0 0 0 0 0 0 0
% N41:20 % 0 2 20002 70 80 98 509 0 0 0
% N41:30 % 0 3 20003 460 0 162 0 0 0 0
% N41:40 % 0 4 20004 120 110 94 508 0 0 0
% N41:50 % 0 5 0 120 110 98 508 0 0 0
% N41:60 % 0 6 20006 230 333 190 0 0 0 0
% N41:70 % 0 7 20005 890 0 275 0 0 0 0
% N41:80 % 0 3 0 370 0 162 0 0 0 0
% N41:90 % 0 9 0 70 30 30 513 0 0 0
% N41:100 % 0 10 0 70 30 30 509 0 0 0
% N41:150 % 0 15 20201 0 0 0 0 0 0 0
DATA N42
% N42:70 % 0 16 0 30 30 20 510 0 0 0
DATA N43
% N43:50 % 0 0 0 0 0 70 0 0 0 0
% N43:100 % 0 0 1 0 1500 100 750 300 300 70
% N43:110 % 15 0 100 0 0 480 0 585 440 650
% N43:120 % 60 30 55 80 30 70 30 95 0 0
% N43:130 % 10 600 0 600 600 600 600 600 300 300
% N43:140 % 300 300 300 0 600 7 40 300 50 60
% N43:150 % 40 60 40 20 5 70 90 20 5 50
% N43:160 % 50 0 0 0 0 0 0 0 0 0
DATA N44
% N44:0 % 0 0 0 0 1500 100 750 300 15 90
% N44:10 % 15 0 100 0 0 800 0 600 800 900
% N44:20 % 60 30 55 60 30 60 30 95 0 0
% N44:30 % 10 600 0 600 600 600 600 600 300 300
% N44:40 % 300 300 300 0 600 30 30 300 50 60
% N44:50 % 40 60 40 5 5 70 30 20 5 50
% N44:60 % 50 0 0 0 0 0 0 0 0 0
% N44:100 % 0 0 1 0 600 100 750 300 300 100
% N44:110 % 15 0 100 0 0 420 0 560 420 650
% N44:120 % 60 30 55 60 30 60 30 95 0 0
% N44:130 % 10 600 0 600 600 600 600 600 300 300
% N44:140 % 300 300 300 0 600 15 30 300 50 60
% N44:150 % 40 60 40 20 5 70 30 20 5 50
% N44:160 % 50 0 0 0 0 0 0 0 0 0
DATA N45
% N45:0 % 0 0 1 0 600 100 750 500 500 75
% N45:10 % 15 0 100 0 0 440 0 550 440 650
% N45:20 % 60 30 55 80 30 70 30 95 0 0
% N45:30 % 10 600 0 600 600 600 600 600 300 300
% N45:40 % 300 300 300 0 600 15 30 300 50 60
% N45:50 % 40 60 40 20 5 70 30 20 5 50
% N45:60 % 50 0 0 0 0 0 0 0 0 0
% N45:100 % 0 0 1 0 1500 100 750 800 300 140
% N45:110 % 20 0 100 0 0 720 0 960 720 900
% N45:120 % 300 30 55 80 30 70 30 95 0 0
% N45:130 % 10 900 0 600 900 900 900 900 300 600
% N45:140 % 600 600 600 0 600 15 30 300 50 60
% N45:150 % 40 60 40 20 5 70 30 20 5 50
% N45:160 % 50 0 0 0 0 0 0 0 0 0
DATA N46
% N46:0 % 0 0 0 0 2250 100 750 300 30 70
% N46:10 % 15 0 100 0 0 1230 0 1140 1230 900
% N46:20 % 60 30 50 60 30 60 30 95 0 0
% N46:30 % 10 600 0 600 600 600 600 600 300 300
% N46:40 % 300 300 300 0 600 15 30 300 50 60
% N46:50 % 40 60 40 10 5 74 30 20 5 50
% N46:60 % 50 0 0 0 0 0 0 0 0 0
DATA N47
% N47:0 % 0 0 1 0 600 0 0 300 300 70
% N47:10 % 15 0 100 0 0 400 0 500 400 300
% N47:20 % 60 30 55 80 30 70 30 95 0 0
% N47:30 % 10 600 0 600 600 600 600 600 300 300
% N47:40 % 300 300 300 0 600 30 40 300 50 60
% N47:50 % 40 60 40 20 5 70 90 20 5 50
% N47:60 % 50 0 0 0 0 0 0 0 0 0
% N47:100 % 0 0 1 0 600 0 0 0 0 0
DATA N50
% N50:100 % 0 0 1 0 1200 100 750 300 300 70
% N50:110 % 15 0 100 0 0 803 0 1005 508 409
% N50:120 % 60 30 50 70 30 60 30 90 0 30
% N50:130 % 10 300 0 120 300 300 300 300 300 300
% N50:140 % 300 300 300 0 120 8 30 120 50 60
% N50:150 % 40 60 40 20 5 70 90 20 5 50
% N50:160 % 50 0 0 0 0 0 0 0 0 0
DATA N60
% N60:0 % 0 2000 800 10 5 5 0 0 480 60
% N60:10 % 480 180 270 135 20 953 0 0 3610 50
% N60:20 % 480 180 500 133 14 858 60 3 0 0
% N60:30 % 1 0 0 0 0 0 0 0 0 0
% N60:50 % 0 60 140 200 150 5 242 80 16 100
% N60:60 % 27 20 20 350 330 2 3 5 5 5
% N60:70 % 5 5 5 0 0 0 0 0 0 0
% N60:100 % 0 2 0 322 0 107 0 0 0 0
% N60:150 % 0 0 0 0 1500 100 750 250 50 70
% N60:160 % 15 0 100 0 0 480 0 444 650 600
% N60:170 % 60 30 50 70 30 60 30 95 0 30
% N60:180 % 10 600 0 600 600 600 600 600 300 300
% N60:190 % 300 300 300 0 600 30 30 300 50 60
% N60:200 % 40 60 40 15 5 74 30 20 5 50
% N60:210 % 50 0 0 0 0 0 0 0 0 0
DATA N61
% N61:0 % 1 0 0 0 0 0 0 0 0 0
% N61:10 % 0 1 20001 414 0 138 0 0 0 0
% N61:20 % 0 2 0 322 0 107 0 0 0 0
% N61:30 % 0 3 0 100 115 88 308 0 0 0
% N61:40 % 0 4 0 100 120 94 308 0 0 0
% N61:50 % 0 5 601 355 0 114 2303 0 0 0
% N61:60 % 0 5 602 355 0 115 0 0 0 0
% N61:70 % 0 5 603 355 0 116 0 0 0 0
% N61:80 % 0 8 604 400 0 0 0 0 0 0
% N61:110 % 0 11 0 152 112 90 10308 0 0 0
DATA N63
% N63:0 % 0 0 0 0 1000 100 750 75 30 250
% N63:10 % 40 0 100 0 0 620 0 630 620 600
% N63:20 % 60 30 50 60 30 60 30 95 0 0
% N63:30 % 10 600 0 600 600 600 600 600 300 300
% N63:40 % 300 300 300 0 600 30 30 300 50 60
% N63:50 % 40 60 40 15 5 74 30 20 5 50
% N63:60 % 50 0 0 0 0 0 0 0 0 0
% N63:100 % 0 0 0 0 1500 100 750 250 50 70
% N63:110 % 15 0 100 0 0 480 0 444 650 600
% N63:120 % 60 30 50 70 30 60 30 95 0 30
% N63:130 % 10 600 0 600 600 600 600 600 300 300
% N63:140 % 300 300 300 0 600 30 30 300 50 60
% N63:150 % 40 60 40 15 5 74 30 20 5 50
% N63:160 % 50 0 0 0 0 0 0 0 0 0
DATA N64
% N64:0 % 0 0 1 0 1000 100 750 500 300 100
% N64:10 % 20 0 100 0 0 600 0 550 600 650
% N64:20 % 60 30 50 70 30 60 30 95 0 0
% N64:30 % 10 600 0 600 600 600 600 600 300 300
% N64:40 % 300 300 300 0 600 5 30 300 50 60
% N64:50 % 40 60 40 20 5 74 30 20 5 50
% N64:60 % 50 0 0 0 0 0 0 0 0 0
% N64:100 % 0 0 1 0 1000 100 750 250 50 200
% N64:110 % 20 0 100 0 0 600 0 550 600 650
% N64:120 % 60 30 50 70 30 60 30 95 0 0
% N64:130 % 10 600 0 600 600 600 600 600 300 300
% N64:140 % 300 300 300 0 600 5 30 300 50 60
% N64:150 % 40 60 40 20 5 74 30 20 5 50
% N64:160 % 50 0 0 0 0 0 0 0 0 0
DATA N65
% N65:0 % 0 0 0 0 1000 100 750 500 500 180
% N65:10 % 50 0 100 0 0 600 0 550 600 700
% N65:20 % 60 30 50 80 30 70 30 95 0 0
% N65:30 % 10 600 0 600 600 600 600 600 300 300
% N65:40 % 300 300 300 0 600 30 30 300 50 60
% N65:50 % 40 60 40 10 5 74 30 20 5 50
% N65:60 % 50 0 0 0 0 0 0 0 0 0
% N65:100 % 0 0 0 0 1000 100 750 500 500 50
% N65:110 % 15 0 100 0 0 515 0 685 515 650
% N65:120 % 60 30 50 80 30 70 30 95 0 30
% N65:130 % 10 600 0 600 600 600 600 600 300 300
% N65:140 % 300 300 300 0 600 30 30 300 50 60
% N65:150 % 40 60 40 5 5 74 30 20 5 50
% N65:160 % 50 0 0 0 0 0 0 0 0 0
DATA N66
% N66:100 % 0 0 0 0 1200 100 750 500 500 240
% N66:110 % 80 0 100 0 0 1165 0 1000 0 669
% N66:120 % 60 30 50 70 30 65 30 95 0 0
% N66:130 % 10 600 0 600 600 600 0 0 0 300
% N66:140 % 300 0 0 0 0 10 10 300 75 65
% N66:150 % 55 60 55 10 6 74 30 20 6 50
% N66:160 % 50 0 0 0 0 0 0 0 0 0
% N66:190 % 0 0 0 0 0 0 0 0 78 24055
DATA N68
% N68:0 % 0 0 1 0 1000 100 750 500 500 50
% N68:10 % 15 0 100 0 0 400 0 530 400 650
% N68:20 % 60 30 50 80 30 70 30 95 0 30
% N68:30 % 10 600 0 600 600 600 600 600 300 300
% N68:40 % 300 300 300 0 600 30 30 300 50 60
% N68:50 % 40 60 40 5 5 74 30 20 5 50
% N68:60 % 50 0 0 0 0 0 0 0 0 0
DATA N80
% N80:0 % 0 1500 800 10 5 5 0 0 1500 60
% N80:10 % 480 180 450 148 15 490 0 0 1500 50
% N80:20 % 480 180 530 133 10 490 60 3 1600 0
% N80:30 % 80 70 0 150 600 300 2000 0 0 0
% N80:50 % 0 90 60 40 100 300 50 300 1 100
% N80:60 % 15 20 20 350 330 2 0 5 5 5
% N80:70 % 5 5 5 3 0 0 0 0 0 0
DATA N100
% N100:0 % 1 1500 0 0 0 0 0 0 0 0
% N100:30 % 0 0 0 0 0 0 1200 0 0 0
% N100:50 % 7807 0 0 0 0 0 0 0 0 0
% N100:60 % 0 384 384 0 0 0 0 0 0 0
% N100:150 % 0 0 0 0 0 100 750 0 0 0
DATA N120
% N120:0 % 0 1500 0 0 0 0 0 0 0 0
% N120:30 % 0 0 0 0 0 0 1200 0 0 0
% N120:100 % 0 0 0 0 0 0 0 31 0 0
% N120:150 % 0 0 0 0 1000 100 750 0 0 0
DATA N140
% N140:0 % 1 1500 0 0 0 0 0 0 0 0
% N140:30 % 0 0 0 0 0 0 1200 0 0 0
% N140:50 % 7807 0 0 0 0 0 0 0 0 0
% N140:60 % 0 384 384 0 0 0 0 0 0 0
% N140:100 % 0 0 0 0 0 0 2817 31 0 0
% N140:150 % 64 0 0 0 1000 100 750 0 0 0
DATA B160
% B160:0 % 0X0002 0X0000 0X0000 0X1200 0X1000 0X0000 0X1800 0X0001 0X2000 0X0000
% B160:10 % 0X0000 0X0000 0X0000 0X0000 0X0000 0X0000 0X0000 0X0000 0X0900 0X0D00
% B160:20 % 0X0006
DATA B161
% B161:0 % 0X0000 0X0000 0X0001 0X0000 0X0000 0X0000 0X0000 0X0000 0X0000 0X0000
% B161:10 % 0X0000 0X0040 0X03C0 0X0000 0X0000 0X0001 0X0000 0X4000 0X2000 0X0000
% B161:20 % 0X0001 0X0100 0X0008 0X0000 0X2080 0X0000 0X0000 0X0000 0X0000 0X0180
% B161:30 % 0X0000 0X0D70 0X0000 0X0000 0X0000 0X0040 0X003F 0X0000 0X0000 0X0000
DATA B162
% B162:0 % 0X0000 0X0000 0X0001 0X0000 0X0000 0X0000 0X0000 0X0000 0X0000 0X0000
% B162:10 % 0X0000 0X0040 0X03C0 0X0000 0X0000 0X0001 0X0000 0X4000 0X0000 0X0000
% B162:20 % 0X0401 0X0100 0X0088 0X0008 0X2080 0X0000 0X0000 0X0000 0X0000 0X0180
% B162:30 % 0X0000 0X0870 0X1881 0X0000 0X0000 0X2040 0X000F 0X0000 0X0000 0X0000
DATA B163
% B163:0 % 0X0000 0X0000 0X0001 0X0000 0X0000 0X0000 0X0000 0X0000 0X0000 0X0000
% B163:10 % 0X0000 0X0040 0X03C0 0X0000 0X0000 0X0000 0X0000 0X4000 0X0080 0X0000
% B163:20 % 0X0401 0X0100 0X8000 0X0000 0X0080 0X0000 0X0000 0X0000 0X0000 0X0180
% B163:30 % 0X3E7F 0X0C70 0X0000 0X0000 0X0000 0X0040 0X0000 0X0000 0X0000 0X0000
DATA B164
% B164:0 % 0X0000 0X0000 0X0001 0X0000 0X0000 0X0000 0X0000 0X0000 0X0000 0X0000
% B164:10 % 0X0000 0X0040 0X03C0 0X0000 0X0000 0X0000 0X0000 0X4000 0X0080 0X0000
% B164:20 % 0X0501 0X0100 0X0008 0X0000 0X0080 0X0000 0X0000 0X0000 0X0000 0X0180
% B164:30 % 0X3E7E 0X0270 0X0000 0X0000 0X0040 0X0060 0X0000 0X0000 0X0000 0X0000
% B164:60 % 0X0000 0X0000 0X0000 0X0000 0X0080 0X0000 0X0000 0X0000 0X0000
DATA B165
% B165:0 % 0X0000 0X0000 0X0001 0X0000 0X0000 0X0000 0X0000 0X0000 0X0000 0X0000
% B165:10 % 0X0000 0X0440 0X03C0 0X0000 0X0000 0X0000 0X0000 0X4000 0X0080 0X0000
% B165:20 % 0X0401 0X0100 0X0008 0X0000 0X0080 0X0000 0X0000 0X0000 0X0000 0X0180
% B165:30 % 0X3E7F 0X0070 0X0000 0X0000 0X0000 0X0040 0X0000 0X0000 0X0000 0X0000
DATA B166
% B166:0 % 0X0000 0X0000 0X0001 0X0000 0X0000 0X0000 0X0000 0X0000 0X0000 0X0000
% B166:10 % 0X0000 0X0040 0X03C0 0X0000 0X0000 0X0000 0X0000 0X480C 0X0000 0X0000
% B166:20 % 0X0401 0X0100 0X0008 0X0000 0X00C0 0X0000 0X0000 0X0000 0X0000 0X2180
% B166:30 % 0X1E7F 0X0010 0X0000 0X0000 0X0040 0X0060 0X0000 0X0000 0X0000 0X0000
% B166:60 % 0X0000 0X0000 0X0000 0X0000 0X2000 0X0000 0X0000 0X0000 0X0000
DATA B169
% B169:0 % 0X0000 0X0000 0X0001 0X0000 0X0000 0X0000 0X0000 0X0000 0X0000 0X0000
% B169:10 % 0X0000 0X0040 0X03C0 0X0000 0X0000 0X0001 0X0000 0X4000 0X0000 0X0000
% B169:20 % 0X0401 0X0100 0X0088 0X0008 0X2090 0X0000 0X0000 0X0000 0X0000 0X0180
% B169:30 % 0X0000 0X0870 0X1881 0X0000 0X0000 0X2040 0X000F 0X0000 0X0000 0X0000
DATA N170
% N170:0 % 222 10601 2 6 0 0 0 0 1 0
% N170:10 % 10 7 7 7 7 7 7 7 10 7
% N170:20 % 7 7 7 7 7 7 3 1 1 1
% N170:50 % 0 105 98 10 3 5 0 20 5 0
% N170:60 % 14 600 2400 1000 4500 4 300 1 4 10
% N170:70 % 20 10 36 2 2 1 1 3 30 90
% N170:80 % 120 150 5 5 105 120 5 30 1800 30
% N170:90 % 35 5 5 2 3600 15 0 600 150 20
% N170:100 % 98 7 3 150 600 2 6 0 0 0
% N170:110 % 0 1 999 1200 0 0 0 211 0 16
% N170:120 % 14 0 6 4 0 2 10 0 0 0
% N170:130 % 0 0 0 0 1 16 1 0 0 0
% N170:200 % 508 509 510 511 512 513 0 0 0 0
DATA N171
% N171:0 % 16512 7 0 0 0 101 0 0 0 0
% N171:20 % 26991 0 10790 10790 0 0 0 0 0 0
% N171:30 % 0 0 0 0 200 1050 1500 1500 1500 291
% N171:40 % 4000 6000 200 23 0 0 0 384 0 0
% N171:50 % 0 0 3440 0 3328 0 0 0 0 0
% N171:80 % 10 0 28 15 350 0 0 0 591 1524
% N171:90 % 0 0 800 0 12286 0 0 0 0 0
% N171:100 % 0 0 0 0 0 0 93 591 591 1
% N171:140 % 401 0 0 0 0 0 0 1 0 63
% N171:150 % 0 4 0 0 0 0 0 0 0 3
% N171:160 % 43 0 -16496 -1 1 0 0 0 0 0
% N171:170 % 108 109 110 111 112 113 0 0 0 0
% N171:200 % 0 0 0 0 0 0 0 0 16495 0
% N171:210 % 0 0 16385 0 0 0 0 0 0 0
% N171:220 % 16495 0 0 0 0 0 0 0 0 0
% N171:230 % 0 6033 5991 3200 6242 6242 0 0
DATA N172
% N172:0 % 16513 7 240 0 0 2 0 0 0 0
% N172:20 % 26992 1 15761 15761 0 0 0 0 0 0
% N172:30 % 0 15 0 0 200 1050 1500 1500 1500 303
% N172:40 % 4000 6000 200 6 0 0 0 384 0 0
% N172:50 % 0 0 2160 0 2064 0 0 0 0 0
% N172:80 % 1 0 28 282 350 0 0 0 591 1524
% N172:90 % 0 0 800 0 10239 0 0 0 0 0
% N172:100 % 0 0 0 0 0 0 115 475 474 1
% N172:140 % 9 0 0 0 0 0 0 128 0 15
% N172:150 % 0 0 0 21 0 0 0 0 0 1
% N172:160 % 41 0 -242 -1 1 0 0 0 0 0
% N172:170 % 308 309 310 311 312 313 0 0 0 0
% N172:200 % 0 0 0 0 0 0 0 0 1 0
% N172:220 % 1 0 0 0 0 0 0 0 0 0
% N172:230 % 32 7551 6228 861 0 0 0 0
DATA N173
% N173:0 % 16513 7 0 0 0 0 0 0 0 0
% N173:20 % 7131 0 5 5 0 0 0 0 0 0
% N173:30 % 0 0 0 0 200 0 1500 1500 1500 132
% N173:40 % 4000 6000 200 1 0 0 15999 384 0 0
% N173:50 % 0 0 3184 0 3120 0 0 0 0 0
% N173:80 % 0 0 0 0 0 0 0 0 1502 2282
% N173:90 % 0 0 0 0 10166 0 0 0 0 0
% N173:120 % 0 0 0 0 0 0 0 0 -15479 0
% N173:140 % 401 0 0 0 0 0 0 0 0 0
% N173:160 % 0 0 -1 -1 0 0 0 0 0 0
% N173:170 % 508 509 510 511 512 513 0 0 0 0
% N173:230 % 2 2542 2720 140 0 0 0 0
DATA N174
% N174:0 % 16513 7 0 0 0 0 0 0 0 0
% N174:20 % 7131 0 98 98 0 0 0 0 0 0
% N174:30 % 0 0 0 0 200 0 1500 1500 1500 113
% N174:40 % 4000 6000 200 0 0 0 15998 384 0 0
% N174:50 % 0 64 624 0 560 0 0 0 0 0
% N174:80 % 0 0 0 0 0 0 0 0 1502 2282
% N174:90 % 0 0 0 0 3927 0 0 0 0 0
% N174:140 % 0 31 0 0 0 0 0 0 0 0
% N174:160 % 0 0 -1 -1 0 0 0 0 0 0
% N174:170 % 708 709 710 711 712 713 0 0 0 0
% N174:230 % 22 2304 2324 0 0 0 0 0
DATA N175
% N175:0 % 16512 7 0 0 0 0 0 0 0 0
% N175:20 % 7132 1 147 147 0 0 0 0 0 0
% N175:30 % 0 0 0 0 200 0 1500 1500 1500 111
% N175:40 % 4000 6000 200 0 0 0 15999 384 0 0
% N175:50 % 0 0 112 0 48 0 0 0 0 0
% N175:80 % 0 0 0 0 0 0 0 0 1502 2282
% N175:90 % 0 0 0 0 4722 0 0 0 0 0
% N175:140 % 0 31 0 0 0 0 0 0 0 0
% N175:160 % 0 0 -1 -1 0 0 0 0 0 0
% N175:170 % 908 909 910 911 912 913 0 0 0 0
% N175:230 % 22 2343 2284 0 0 0 0 0
DATA N176
% N176:0 % 16513 7 0 0 0 0 0 0 0 0
% N176:20 % 7132 1 364 364 0 0 0 0 0 0
% N176:30 % 0 0 0 0 200 0 1500 1500 1500 109
% N176:40 % 4000 6000 200 0 0 0 7807 8576 0 0
% N176:50 % 0 64 16 0 16 0 0 0 0 0
% N176:80 % 0 0 0 0 0 0 0 0 1502 2282
% N176:90 % 0 0 0 0 3670 0 0 0 0 0
% N176:140 % 0 31 0 0 0 0 0 0 0 0
% N176:160 % 0 0 -1 -1 0 0 0 0 0 0
% N176:170 % 1108 1109 1110 1111 1112 1113 0 0 0 0
% N176:230 % 12 2264 2254 0 0 0 0 0
DATA N179
% N179:0 % 16512 7 0 0 0 101 0 0 0 0
% N179:20 % 26995 0 10790 10790 0 0 0 0 0 0
% N179:30 % 0 0 0 0 200 1050 1500 1500 1500 291
% N179:40 % 4000 6000 200 6 0 0 0 384 0 0
% N179:50 % 0 0 2160 0 2064 0 0 0 0 0
% N179:80 % 1 0 28 282 350 0 0 0 591 1524
% N179:90 % 0 0 800 0 10239 0 0 0 0 0
% N179:100 % 0 0 0 0 0 0 115 475 474 1
% N179:140 % 9 0 0 0 0 0 0 128 0 15
% N179:150 % 0 0 0 21 0 0 0 0 0 1
% N179:160 % 41 0 -242 -1 1 0 0 0 0 0
% N179:170 % 308 309 310 311 312 313 0 0 0 0
% N179:200 % 0 0 0 0 0 0 0 0 1 0
% N179:220 % 1 0 0 0 0 0 0 0 0 0
% N179:230 % 12 7551 6228 871 0 0 0 0
DATA T180
% .PRE .ACC %
% T180:0 % 60 0
% T180:1 % 30 43
% T180:2 % 200 0
% T180:3 % 32767 26996
% T180:4 % 20 0
% T180:5 % 2 0
% T180:6 % 7 0
DATA T181
% .PRE .ACC %
% T181:0 % 5 0
% T181:1 % 300 0
% T181:2 % 900 0
% T181:3 % 30 0
% T181:4 % 200 0
% T181:5 % 110 113
% T181:6 % 200 201
% T181:7 % 200 204
% T181:8 % 200 203
% T181:9 % 200 200
% T181:10 % 200 200
% T181:11 % 110 113
% T181:12 % 0 7
% T181:13 % 3 0
% T181:14 % 30 0
% T181:15 % 120 0
% T181:16 % 3 3
% T181:17 % 1 0
% T181:18 % 1 1
% T181:20 % 10 0
% T181:21 % 30 0
% T181:22 % 10 0
% T181:23 % 1 1
% T181:24 % 8 37
% T181:26 % 4 0
% T181:27 % 2 0
% T181:28 % 3 0
% T181:29 % 5 0
% T181:30 % 3 0
% T181:31 % 2 0
% T181:32 % 2 0
% T181:33 % 50 57
% T181:34 % 3 0
% T181:36 % 10 0
% T181:37 % 7 0
% T181:38 % 7 0
% T181:39 % 7 0
% T181:40 % 7 0
% T181:41 % 7 0
% T181:42 % 7 0
% T181:43 % 7 0
% T181:44 % 10 0
% T181:45 % 7 0
% T181:46 % 7 0
% T181:47 % 7 0
% T181:48 % 7 0
% T181:49 % 7 0
% T181:50 % 7 0
% T181:51 % 7 0
% T181:52 % 3 0
% T181:53 % 1 0
% T181:54 % 1 0
% T181:55 % 1 0
% T181:56 % 3 0
% T181:57 % 3 0
% T181:58 % 3 0
% T181:59 % 3 0
% T181:60 % 3 0
% T181:61 % 3 0
% T181:62 % 3 0
% T181:63 % 3 0
% T181:64 % 32767 0
% T181:65 % 15 0
% T181:66 % 200 200
DATA T182
% .PRE .ACC %
% T182:0 % 5 0
% T182:1 % 300 0
% T182:2 % 600 0
% T182:3 % 30 0
% T182:4 % 200 0
% T182:5 % 110 110
% T182:6 % 200 207
% T182:7 % 200 203
% T182:8 % 200 204
% T182:9 % 200 200
% T182:10 % 200 200
% T182:11 % 110 110
% T182:12 % 0 7
% T182:13 % 3 0
% T182:14 % 30 0
% T182:15 % 140 0
% T182:16 % 3 3
% T182:17 % 1 1
% T182:18 % 1 1
% T182:19 % 8 0
% T182:20 % 10 0
% T182:21 % 30 30
% T182:22 % 10 0
% T182:23 % 1 1
% T182:24 % 4 0
% T182:26 % 4 0
% T182:27 % 2 0
% T182:28 % 20 0
% T182:29 % 5 0
% T182:30 % 3 0
% T182:31 % 3 0
% T182:32 % 3 0
% T182:33 % 50 50
% T182:34 % 3 0
% T182:36 % 10 0
% T182:37 % 7 0
% T182:38 % 7 0
% T182:39 % 7 0
% T182:40 % 7 0
% T182:41 % 7 0
% T182:42 % 7 0
% T182:43 % 7 0
% T182:44 % 10 0
% T182:45 % 7 0
% T182:46 % 7 0
% T182:47 % 7 0
% T182:48 % 7 0
% T182:49 % 7 0
% T182:50 % 7 0
% T182:51 % 7 0
% T182:52 % 3 0
% T182:53 % 1 0
% T182:54 % 1 0
% T182:55 % 1 0
% T182:56 % 3 0
% T182:57 % 3 0
% T182:58 % 3 0
% T182:59 % 3 0
% T182:60 % 3 0
% T182:61 % 3 0
% T182:62 % 3 0
% T182:63 % 3 0
% T182:64 % 32767 0
% T182:65 % 15 0
% T182:66 % 200 200
DATA T183
% .PRE .ACC %
% T183:0 % 5 0
% T183:3 % 64 0
% T183:4 % 200 0
% T183:5 % 110 114
% T183:6 % 200 200
% T183:7 % 200 200
% T183:8 % 200 200
% T183:9 % 200 200
% T183:10 % 200 200
% T183:11 % 110 114
% T183:12 % 0 6
% T183:16 % 3 3
% T183:17 % 2 0
% T183:18 % 2 2
% T183:20 % 10 0
% T183:22 % 10 0
% T183:23 % 1 1
% T183:27 % 2 0
% T183:28 % 200 0
% T183:29 % 3 0
% T183:30 % 3 0
% T183:31 % 3 0
% T183:32 % 3 0
% T183:33 % 50 57
% T183:34 % 3 0
% T183:36 % 10 0
% T183:37 % 7 0
% T183:38 % 7 0
% T183:39 % 7 0
% T183:40 % 7 0
% T183:41 % 7 0
% T183:42 % 7 0
% T183:43 % 7 0
% T183:44 % 10 0
% T183:45 % 7 0
% T183:46 % 7 0
% T183:47 % 7 0
% T183:48 % 7 0
% T183:49 % 7 0
% T183:50 % 7 0
% T183:51 % 7 0
% T183:52 % 3 0
% T183:53 % 1 0
% T183:54 % 1 0
% T183:55 % 1 0
% T183:56 % 3 0
% T183:57 % 3 0
% T183:58 % 3 0
% T183:59 % 3 0
% T183:60 % 3 0
% T183:61 % 3 0
% T183:62 % 3 0
% T183:63 % 3 0
% T183:64 % 32767 0
% T183:65 % 15 0
% T183:66 % 200 200
DATA T184
% .PRE .ACC %
% T184:0 % 200 0
% T184:3 % 64 0
% T184:4 % 200 0
% T184:5 % 110 114
% T184:6 % 200 200
% T184:7 % 200 200
% T184:8 % 200 200
% T184:9 % 200 200
% T184:10 % 200 200
% T184:11 % 110 114
% T184:12 % 0 6
% T184:16 % 3 0
% T184:17 % 1 1
% T184:18 % 200 0
% T184:22 % 10 0
% T184:23 % 1 1
% T184:28 % 200 0
% T184:29 % 3 0
% T184:30 % 3 0
% T184:31 % 3 0
% T184:32 % 3 0
% T184:33 % 50 57
% T184:34 % 3 0
% T184:36 % 10 0
% T184:37 % 7 0
% T184:38 % 7 0
% T184:39 % 7 0
% T184:40 % 7 0
% T184:41 % 7 0
% T184:42 % 7 0
% T184:43 % 7 0
% T184:44 % 10 0
% T184:45 % 7 0
% T184:46 % 7 0
% T184:47 % 7 0
% T184:48 % 7 0
% T184:49 % 7 0
% T184:50 % 7 0
% T184:51 % 7 0
% T184:52 % 3 0
% T184:53 % 1 0
% T184:54 % 1 0
% T184:55 % 1 0
% T184:56 % 3 0
% T184:57 % 3 0
% T184:58 % 3 0
% T184:59 % 3 0
% T184:60 % 3 0
% T184:61 % 3 0
% T184:62 % 3 0
% T184:63 % 3 0
% T184:64 % 32767 0
% T184:65 % 15 0
% T184:66 % 200 200
DATA T185
% .PRE .ACC %
% T185:0 % 200 0
% T185:4 % 200 0
% T185:5 % 110 114
% T185:6 % 200 200
% T185:7 % 200 200
% T185:8 % 200 200
% T185:9 % 200 200
% T185:10 % 200 200
% T185:11 % 110 114
% T185:12 % 0 6
% T185:16 % 3 3
% T185:17 % 1 1
% T185:18 % 200 0
% T185:22 % 10 0
% T185:23 % 1 1
% T185:28 % 200 0
% T185:29 % 3 0
% T185:30 % 3 0
% T185:31 % 3 0
% T185:32 % 3 0
% T185:33 % 50 57
% T185:34 % 3 0
% T185:36 % 10 0
% T185:37 % 7 0
% T185:38 % 7 0
% T185:39 % 7 0
% T185:40 % 7 0
% T185:41 % 7 0
% T185:42 % 7 0
% T185:43 % 7 0
% T185:44 % 10 0
% T185:45 % 7 0
% T185:46 % 7 0
% T185:47 % 7 0
% T185:48 % 7 0
% T185:49 % 7 0
% T185:50 % 7 0
% T185:51 % 7 0
% T185:52 % 3 0
% T185:53 % 1 0
% T185:54 % 1 0
% T185:55 % 1 0
% T185:56 % 3 0
% T185:57 % 3 0
% T185:58 % 3 0
% T185:59 % 3 0
% T185:60 % 3 0
% T185:61 % 3 0
% T185:62 % 3 0
% T185:63 % 3 0
% T185:64 % 32767 0
% T185:65 % 15 0
% T185:66 % 200 200
DATA T186
% .PRE .ACC %
% T186:0 % 200 0
% T186:3 % 64 0
% T186:4 % 200 0
% T186:5 % 110 114
% T186:6 % 200 200
% T186:7 % 200 200
% T186:8 % 200 200
% T186:9 % 200 200
% T186:10 % 200 200
% T186:11 % 110 114
% T186:12 % 0 6
% T186:16 % 3 3
% T186:17 % 1 1
% T186:18 % 200 0
% T186:22 % 10 0
% T186:23 % 1 1
% T186:29 % 3 0
% T186:30 % 3 0
% T186:31 % 3 0
% T186:32 % 3 0
% T186:33 % 50 57
% T186:34 % 3 0
% T186:36 % 10 0
% T186:37 % 7 0
% T186:38 % 7 0
% T186:39 % 7 0
% T186:40 % 7 0
% T186:41 % 7 0
% T186:42 % 7 0
% T186:43 % 7 0
% T186:44 % 10 0
% T186:45 % 7 0
% T186:46 % 7 0
% T186:47 % 7 0
% T186:48 % 7 0
% T186:49 % 7 0
% T186:50 % 7 0
% T186:51 % 7 0
% T186:52 % 3 0
% T186:53 % 1 0
% T186:54 % 1 0
% T186:55 % 1 0
% T186:56 % 3 0
% T186:57 % 3 0
% T186:58 % 3 0
% T186:59 % 3 0
% T186:60 % 3 0
% T186:61 % 3 0
% T186:62 % 3 0
% T186:63 % 3 0
% T186:64 % 32767 0
% T186:65 % 15 0
% T186:66 % 200 200
DATA N191
% N191:0 % 19 0 0 300 15 0 0 0 0 0
% N191:10 % 0 0 0 30 0 0 0 0 0 0
% N191:20 % 0 0 0 3205 0 293 0 0 0 0
% N191:40 % 27 0 0 90 15 0 0 0 0 0
% N191:50 % 0 100 0 30 0 0 0 0 0 0
% N191:60 % 0 0 0 5 0 1 0 0 0 0
DATA N192
% N192:0 % 19 0 0 250 50 0 0 0 0 0
% N192:10 % 0 0 0 30 0 0 0 0 0 0
% N192:20 % 0 0 0 4011 0 367 0 0 0 0
% N192:40 % 27 0 0 70 15 0 0 0 0 0
% N192:50 % 0 100 0 30 0 0 0 0 0 0
% N192:60 % 0 0 0 12 0 3 0 0 0 0
DATA N193
% N193:0 % 19 0 0 100 5 0 0 0 0 0
% N193:10 % 0 0 0 30 0 0 0 0 0 0
% N193:20 % 0 0 0 1356 0 124 0 0 0 0
% N193:40 % 27 0 0 50 5 0 0 0 0 0
% N193:50 % 0 100 1 30 0 0 0 0 0 0
% N193:60 % 0 0 0 1 0 0 0 0 0 0
DATA N194
% N194:0 % 1 0 0 0 0 0 0 0 0 0
% N194:10 % 0 0 0 30 0 0 0 0 0 0
% N194:20 % 0 0 0 1224 0 112 0 0 0 0
% N194:40 % 27 0 0 0 0 0 0 0 0 0
% N194:50 % 0 0 0 30 0 0 0 0 0 0
% N194:60 % 0 0 0 1 0 0 0 0 0 0
DATA N195
% N195:0 % 19 0 0 0 0 0 0 0 0 0
% N195:10 % 0 0 0 30 0 0 0 0 0 0
% N195:20 % 0 0 0 1245 0 114 0 0 0 0
% N195:40 % 27 0 0 0 0 0 0 0 0 0
% N195:50 % 0 0 0 30 0 0 0 0 0 0
% N195:60 % 0 0 0 12 0 3 0 0 0 0
DATA N196
% N196:0 % 19 0 0 0 0 0 0 0 0 0
% N196:10 % 0 0 0 30 0 0 0 0 0 0
% N196:20 % 0 0 0 1203 0 110 0 0 0 0
% N196:40 % 27 0 0 0 0 0 0 0 0 0
% N196:50 % 0 0 0 30 0 0 0 0 0 0
% N196:60 % 0 0 0 12 0 3 0 0 0 0
DATA N200
% N200:20 % 0 1 0 0 0 0 0 0 0 0
% N200:40 % 0 26 0 0 0 0 0 0 0 0
DATA N201
% N201:10 % 0 0 0 0 0 0 12286
DATA N202
% N202:10 % 0 0 0 0 0 0 10239
DATA N203
% N203:10 % 0 0 0 0 0 0 10167
DATA N204
% N204:10 % 0 0 0 0 0 0 3930
DATA N205
% N205:10 % 0 0 0 0 0 0 4725
DATA N206
% N206:10 % 0 0 0 0 0 0 3673
DATA N211
% N211:0 % 0 2 -4076 1088 84 0 0 0 0 0
% N211:10 % 0 0 0 0 0 0 -16496 -1 0 0
% N211:30 % 0 293 0 291 0 23 0 0 0 0
% N211:40 % 0 0 3673
DATA N212
% N212:0 % 0 2 -4076 1088 84 0 0 0 0 0
% N212:10 % 0 0 0 0 0 0 -242 -1 0 0
% N212:30 % 0 367 0 303 0 6 0 0 0 0
% N212:40 % 0 0 3673
DATA N213
% N213:0 % 0 2 -4076 32 68 0 0 0 0 0
% N213:10 % 0 0 0 0 0 0 -1 -1 0 0
% N213:30 % 0 124 0 132 0 1 0 0 0 15999
% N213:40 % 0 0 3932
DATA N214
% N214:0 % 0 2 -4076 72 0 0 0 0 0 0
% N214:10 % 128 0 0 0 0 0 -1 -1 0 0
% N214:30 % 0 112 0 113 0 0 0 0 0 15998
% N214:40 % 0 0 3932
DATA N215
% N215:0 % 0 2 -4076 64 68 0 0 0 0 0
% N215:10 % 0 0 0 0 0 0 -1 -1 0 0
% N215:30 % 0 114 0 111 0 0 0 0 0 15999
% N215:40 % 0 0 3932
DATA N216
% N216:0 % 0 -32767 -4092 72 68 0 0 0 0 0
% N216:10 % 8192 0 0 0 0 0 -1 -1 0 0
% N216:30 % 0 110 0 109 0 0 0 0 0 7807
% N216:40 % 0 0 3675
DATA N231
% N231:40 % 0 353 256 256 256 256 256 0 0 0
DATA N232
% N232:0 % 0 129 0 0 0 0 0 0 0 0
% N232:40 % 0 256 256 256 256 0 0 0 0 0
